Fanuc KAREL source: kt00492.KL

-- PROVISIONAL review KL for V770-1; original PC SHA256 56ad2fceab303ae5409b24b566e650c2294137b2de2adcb9e1fd4144b57340fa
-- Incomplete behavior may be omitted. Consult companion uncertainty JSON. Do not deploy.
PROGRAM KT00492
%NOLOCKGROUP
-- UNRESOLVED_DECL P1 type=000101
-- UNRESOLVED_DECL P2 type=000199
-- UNRESOLVED_DECL OUT type=000199
BEGIN
  -- UNRESOLVED_PC offsets 5-39; opcodes 49,49,7E,60,7E,4A
  -- UNRESOLVED_PC offsets 44-48; opcodes 7F
END KT00492
